FUNCTION_BLOCK FB_ValveOutput
VAR_INPUT
	bEnable 			: BOOL;
	stValveDeadBand 	: ST_ValveDeadBand;
	fNormalizedInput 	: LREAL;
END_VAR
VAR_OUTPUT
	bEnableValveOutput : BOOL;
	nOutput : INT; 
END_VAR
VAR
	nOffset 	: INT := 19660;
	nMaxValue	: INT := 29490;
	nMinValue 	: INT :=  9830;
	nTempOutput : INT;
END_VAR

IF fNormalizedInput > 0.0 THEN
	nTempOutput := LREAL_TO_INT(ABS(fNormalizedInput*(stValveDeadBand.fPosMax - stValveDeadBand.fPosMin) + stValveDeadBand.fPosMin));
ELSIF fNormalizedInput < 0.0 THEN
	nTempOutput := LREAL_TO_INT(ABS(fNormalizedInput*(stValveDeadBand.fNegMax - stValveDeadBand.fNegMin) - stValveDeadBand.fNegMin));
ELSE
	nTempOutput := nOffset;
END_IF

IF NOT(bEnable) THEN
	nOutput := nOffset;
	bEnableValveOutput := FALSE;
ELSE
	nOutput := LIMIT(nMinValue, nTempOutput, nMaxValue);
	bEnableValveOutput := TRUE; 
END_IF

END_FUNCTION_BLOCK

(* stored: Version 1.1.0.1, ProductVersion 3.1.4024.11
   POU FB_ValveOutput: Id {f59c2bfb-80b3-4afa-9ddc-65e6b1ad119e}, SpecialFunc None *)
